{attribute addProperty BoxType "EM7004-0000-0017"}
{attribute addProperty Id "InputAT %I*Input_D06BCD81162"}
{attribute addProperty CRC "4157845918"}
{attribute addProperty SizeInBites "16"}
{attribute addProperty SizeInBytes "2"}
TYPE DI_Inputs_F7D3B19E :
STRUCT
	{attribute addProperty Name "Input"}
	Input AT %I* : Input_D06BCD81;
END_STRUCT
END_TYPE

(* stored: Version 1.2.0.0, ProductVersion 3.1.4024.9
   DUT DI_Inputs_F7D3B19E: Id {e0b7aa8c-23d5-446d-8284-24cd10a19c17} *)
